PROGRAM PRG_StoppedState
VAR
	fbBlinkStartButton	:	FB_Blink;
END_VAR

//Start Button Blink ------------------------------------------------
IF GVL_Safety.bSafetyEnable AND NOT GVL_HMI.bIncoherenceDetected THEN
	fbBlinkStartButton( bEnable := TRUE, tPeriod := T#1S );
ELSE
	fbBlinkStartButton( bEnable := FALSE, tPeriod := T#1S );
END_IF

GVL_IO.gDigOutputs.bStartIndicator := fbBlinkStartButton.bBlink;

END_PROGRAM

(* stored: Version 1.1.0.1, ProductVersion 3.1.4024.12
   POU PRG_StoppedState: Id {e1a020b0-65f1-4f8b-82e2-3f08dab3c53c}, SpecialFunc None *)
